PROGRAM MAIN
VAR
	
	fbConveyor : FB_Conveyor;
	iConveyor : I_Conveyor;
END_VAR

iConveyor := fbConveyor;

END_PROGRAM

(* stored: Version 1.1.0.1, ProductVersion 3.1.4024.16
   POU MAIN: Id {35a7ba89-cc06-46c8-9519-2cb750099650}, SpecialFunc None *)
